// SIMATIC S7-200 SMART project (STEP 7-Micro/WIN SMART), CPU ST60

SYMBOL_TABLE Table 1
GLASS_SUCK       M10.1
AUTO_COIL        M10.0
CYL_DN_MEM_BITS  M0.7
READY_COIL       M0.6
REV_COIL         M0.5
FAWARD_COIL      M0.4
SUCK_COIL        M0.3
AUTO_SEL         M0.1
MAN_SEL          M0.0
END_SYMBOL_TABLE

SYMBOL_TABLE System Symbols
Always_On        SM0.0    // Always ON
END_SYMBOL_TABLE

ORGANIZATION_BLOCK MAIN:OB1
TITLE=MHSF 
BEGIN
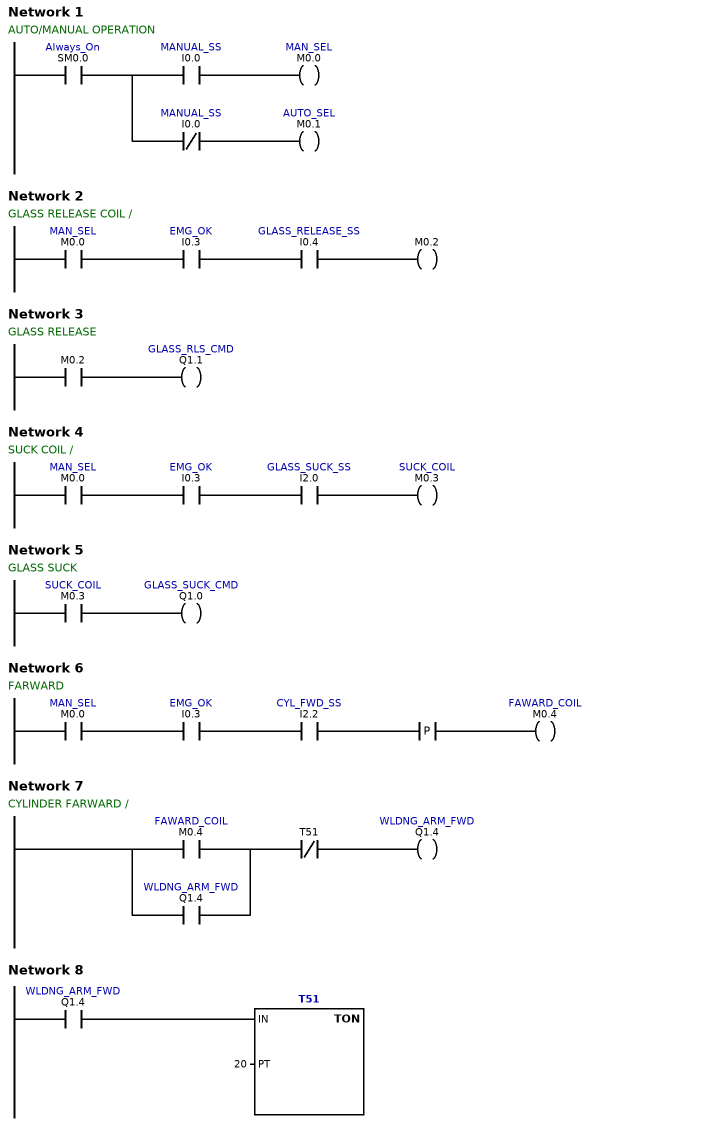
Network 1
// AUTO/MANUAL OPERATION 
LD     Always_On:SM0.0
LPS
A      MANUAL_SS:I0.0
=      MAN_SEL:M0.0
LPP
AN     MANUAL_SS:I0.0
=      AUTO_SEL:M0.1
Network 2
// GLASS RELEASE COIL
// 
LD     MAN_SEL:M0.0
A      EMG_OK:I0.3
A      GLASS_RELEASE_SS:I0.4
=      M0.2
Network 3
// GLASS RELEASE
LD     M0.2
=      GLASS_RLS_CMD:Q1.1
Network 4
// SUCK COIL
// 
LD     MAN_SEL:M0.0
A      EMG_OK:I0.3
A      GLASS_SUCK_SS:I2.0
=      SUCK_COIL:M0.3
Network 5
// GLASS SUCK
LD     SUCK_COIL:M0.3
=      GLASS_SUCK_CMD:Q1.0
Network 6
// FARWARD
LD     MAN_SEL:M0.0
A      EMG_OK:I0.3
A      CYL_FWD_SS:I2.2
EU
=      FAWARD_COIL:M0.4
Network 7
// CYLINDER FARWARD
// 
// (network saved uncompiled; LAD cells follow)
// row 0: c0 -- v  c1 -| |- FAWARD_COIL:M0.4 v  c2 -|/|- T51  c3 -( ) WLDNG_ARM_FWD:Q1.4
// row 1: c0 ^  c1 -| |- WLDNG_ARM_FWD:Q1.4 ^
Network 8
LD     WLDNG_ARM_FWD:Q1.4
TON    T51, 20
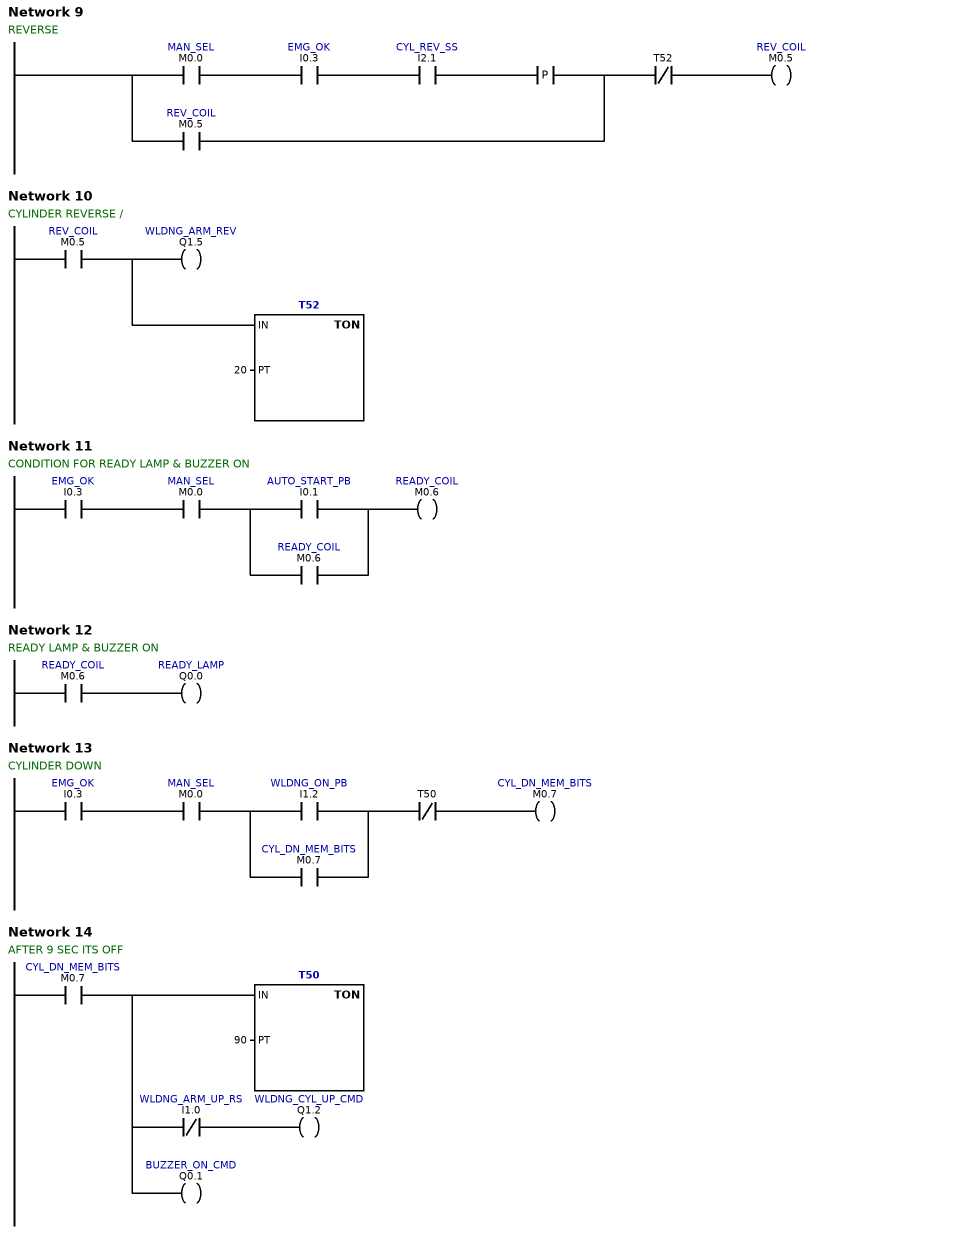
Network 9
// REVERSE
// (network saved uncompiled; LAD cells follow)
// row 0: c0 -- v  c1 -| |- MAN_SEL:M0.0  c2 -| |- EMG_OK:I0.3  c3 -| |- CYL_REV_SS:I2.1  c4 -|P|-  v  c5 -|/|- T52  c6 -( ) REV_COIL:M0.5
// row 1: c0 ^  c1 -| |- REV_COIL:M0.5  c2 --  c3 --  c4 -- ^
Network 10
// CYLINDER REVERSE
// 
LD     REV_COIL:M0.5
=      WLDNG_ARM_REV:Q1.5
TON    T52, 20
Network 11
// CONDITION FOR READY LAMP & BUZZER ON
LD     EMG_OK:I0.3
A      MAN_SEL:M0.0
LD     AUTO_START_PB:I0.1
O      READY_COIL:M0.6
ALD
=      READY_COIL:M0.6
Network 12
// READY LAMP & BUZZER ON 
LD     READY_COIL:M0.6
=      READY_LAMP:Q0.0
Network 13
// CYLINDER DOWN 
LD     EMG_OK:I0.3
A      MAN_SEL:M0.0
LD     WLDNG_ON_PB:I1.2
O      CYL_DN_MEM_BITS:M0.7
ALD
AN     T50
=      CYL_DN_MEM_BITS:M0.7
Network 14
// AFTER 9 SEC ITS OFF
LD     CYL_DN_MEM_BITS:M0.7
LPS
TON    T50, 90
AN     WLDNG_ARM_UP_RS:I1.0
=      WLDNG_CYL_UP_CMD:Q1.2
LPP
=      BUZZER_ON_CMD:Q0.1
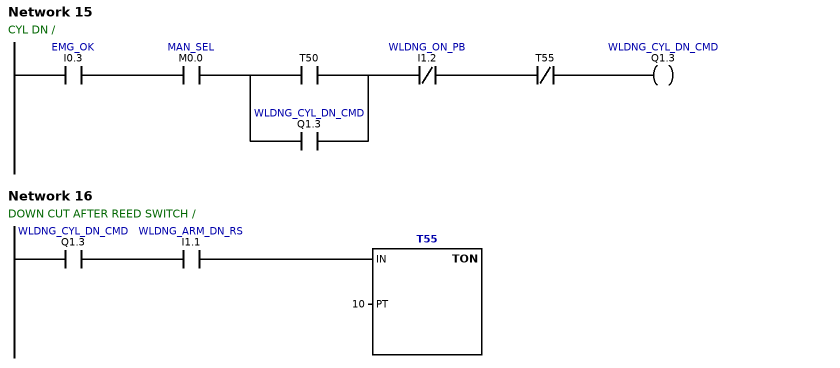
Network 15
// CYL DN
// 
LD     EMG_OK:I0.3
A      MAN_SEL:M0.0
LD     T50
O      WLDNG_CYL_DN_CMD:Q1.3
ALD
AN     WLDNG_ON_PB:I1.2
AN     T55
=      WLDNG_CYL_DN_CMD:Q1.3
Network 16
// DOWN CUT AFTER REED SWITCH
// 
LD     WLDNG_CYL_DN_CMD:Q1.3
A      WLDNG_ARM_DN_RS:I1.1
TON    T55, 10
END_ORGANIZATION_BLOCK
